FUNCTION_BLOCK Plant_SMV (* Composite Function Block Type *)
  (* Standard: 61499-2 *)
  (* Version 0.2, 2003-12-05, JHC, Rockwell Automation, Renamed from NEWCOMPFB. *)
  (* Version 0.1, 2002-01-08, JHC, Rockwell Automation, Added DLY FB as example. *)
  (* Version 0.0, 2000-05-27, JHC, Rockwell Automation *)
  (* Compiler header: package fb.rt.pnp; *)
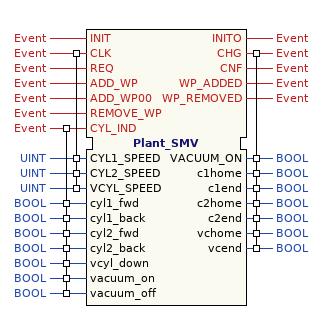
  EVENT_INPUT
    INIT; (* Initialization Request *)
    CLK WITH CYL1_SPEED, CYL2_SPEED, VCYL_SPEED; (* Clock *)
    REQ;
    ADD_WP;
    ADD_WP00;
    REMOVE_WP;
    CYL_IND WITH cyl1_fwd, cyl1_back, cyl2_fwd, cyl2_back, vcyl_down, vacuum_on, vacuum_off;
  END_EVENT
  EVENT_OUTPUT
    INITO; (* Initialization Confirm *)
    CHG WITH c1home, c1end, c2home, c2end, vchome, vcend, VACUUM_ON; (* View State Changed *)
    CNF;
    WP_ADDED;
    WP_REMOVED;
  END_EVENT
  VAR_INPUT
    CYL1_SPEED : UINT;
    CYL2_SPEED : UINT;
    VCYL_SPEED : UINT;
    cyl1_fwd : BOOL;
    cyl1_back : BOOL; (* Response Data from Socket *)
    cyl2_fwd : BOOL;
    cyl2_back : BOOL;
    vcyl_down : BOOL;
    vacuum_on : BOOL;
    vacuum_off : BOOL;
  END_VAR
  VAR_OUTPUT
    VACUUM_ON : BOOL; (* Response Data from Socket *)
    c1home : BOOL;
    c1end : BOOL;
    c2home : BOOL;
    c2end : BOOL;
    vchome : BOOL;
    vcend : BOOL;
  END_VAR
  FBS
    Cylinder : PnpCylinders(InitialPosition := 0.0, HomeSensorRange := [0,0], MidSensorRange := [50,50], EndSensorRange := [100,100], Loaded := 0, LoadType := 0, LCMovingtDistance := 75, RCMovingtDistance := 150, VCMovingtDistance := 75);
    SuctionUnit : PnPVacuum;
  END_FBS
  EVENT_CONNECTIONS
    INIT TO Cylinder.INIT;
    Cylinder.INITO TO SuctionUnit.INIT;
    CLK TO Cylinder.CLK;
    CYL_IND TO Cylinder.CYL_IND;
    CYL_IND TO SuctionUnit.CLK;
    Cylinder.CHG TO CHG;
    SuctionUnit.CHG TO CHG;
  END_CONNECTIONS
  DATA_CONNECTIONS
    CYL1_SPEED TO Cylinder.LCForwardSpeed;
    CYL1_SPEED TO Cylinder.LCBackwardSpeed;
    CYL2_SPEED TO Cylinder.RCForwardSpeed;
    CYL2_SPEED TO Cylinder.RCBackwardSpeed;
    VCYL_SPEED TO Cylinder.VCSpeed;
    cyl1_fwd TO Cylinder.LCExtend;
    cyl1_back TO Cylinder.LCRetract;
    cyl2_fwd TO Cylinder.RCExtend;
    cyl2_back TO Cylinder.RCRetract;
    vcyl_down TO Cylinder.VCExtend;
    Cylinder.LCAtHome TO c1home;
    Cylinder.LCAtEnd TO c1end;
    Cylinder.RCAtHome TO c2home;
    Cylinder.RCAtEnd TO c2end;
    Cylinder.VCAtHome TO vchome;
    Cylinder.VCAtEnd TO vcend;
    SuctionUnit.VacState TO VACUUM_ON;
    vacuum_on TO SuctionUnit.VacuumOn;
    vacuum_off TO SuctionUnit.VacuumOff;
  END_CONNECTIONS
END_FUNCTION_BLOCK
